# EPICS autosave request: displayIOC/autoSaveRestore/display_settings.req
$(P)TriggerDelayAbs
$(P)TriggerMode

$(P)$(CAM1):DISP_MAX
$(P)$(CAM1):OVER_X
$(P)$(CAM1):OVER_Y
$(P)$(CAM1):OVER_SIZE
$(P)$(CAM1):OVER_WIDTH
$(P)$(CAM1):ROI_X
$(P)$(CAM1):ROI_W
$(P)$(CAM1):ROI_Y
$(P)$(CAM1):ROI_H

$(P)$(CAM2):DISP_MAX
$(P)$(CAM2):OVER_X
$(P)$(CAM2):OVER_Y
$(P)$(CAM2):OVER_SIZE
$(P)$(CAM2):OVER_WIDTH
$(P)$(CAM2):ROI_X
$(P)$(CAM2):ROI_W
$(P)$(CAM2):ROI_Y
$(P)$(CAM2):ROI_H

$(P)$(CAM3):DISP_MAX
$(P)$(CAM3):OVER_X
$(P)$(CAM3):OVER_Y
$(P)$(CAM3):OVER_SIZE
$(P)$(CAM3):OVER_WIDTH
$(P)$(CAM3):ROI_X
$(P)$(CAM3):ROI_W
$(P)$(CAM3):ROI_Y
$(P)$(CAM3):ROI_H

$(P)$(CAM4):DISP_MAX
$(P)$(CAM4):OVER_X
$(P)$(CAM4):OVER_Y
$(P)$(CAM4):OVER_SIZE
$(P)$(CAM4):OVER_WIDTH
$(P)$(CAM4):ROI_X
$(P)$(CAM4):ROI_W
$(P)$(CAM4):ROI_Y
$(P)$(CAM4):ROI_H

$(P)$(CAM5):DISP_MAX
$(P)$(CAM5):OVER_X
$(P)$(CAM5):OVER_Y
$(P)$(CAM5):OVER_SIZE
$(P)$(CAM5):OVER_WIDTH
$(P)$(CAM5):ROI_X
$(P)$(CAM5):ROI_W
$(P)$(CAM5):ROI_Y
$(P)$(CAM5):ROI_H

$(P)$(CAM6):DISP_MAX
$(P)$(CAM6):OVER_X
$(P)$(CAM6):OVER_Y
$(P)$(CAM6):OVER_SIZE
$(P)$(CAM6):OVER_WIDTH
$(P)$(CAM6):ROI_X
$(P)$(CAM6):ROI_W
$(P)$(CAM6):ROI_Y
$(P)$(CAM6):ROI_H

$(P)$(CAM7):DISP_MAX
$(P)$(CAM7):OVER_X
$(P)$(CAM7):OVER_Y
$(P)$(CAM7):OVER_SIZE
$(P)$(CAM7):OVER_WIDTH
$(P)$(CAM7):ROI_X
$(P)$(CAM7):ROI_W
$(P)$(CAM7):ROI_Y
$(P)$(CAM7):ROI_H

$(P)$(CAM8):DISP_MAX
$(P)$(CAM8):OVER_X
$(P)$(CAM8):OVER_Y
$(P)$(CAM8):OVER_SIZE
$(P)$(CAM8):OVER_WIDTH
$(P)$(CAM8):ROI_X
$(P)$(CAM8):ROI_W
$(P)$(CAM8):ROI_Y
$(P)$(CAM8):ROI_H

$(P)NF_E_CAL
$(P)PMP_T_E_CAL
$(P)PMP_R_E_CAL
